// SIMATIC STEP 7 (V5.x) project Сварная машина 1
// CPU: CPU 316-2 DP
// station: Hardware
// station: SIMATIC 300(1)
// station: P_ADR_BUS
// station: P_ADR_BUS
// station: Configuration

SYMBOL_TABLE
"C1"	C 1	COUNTER	// Счетчик единиц
"C2"	C 2	COUNTER	// Счетчик тысяч
"C3"	C 3	COUNTER	// Счетчик миллионов
"FC1"	FC 1	FC 1	// Блокировки
"FC2"	FC 2	FC 2	// Управление транспортерами и вентиляторами
"FC3"	FC 3	FC 3	// Муфта
"FC4"	FC 4	FC 4	// Протяжка проволоки
"FC5"	FC 5	FC 5	// Регулировка скорости
"FC6"	FC 6	FC 6	// Привод сварной машины
"FC7"	FC 7	FC 7
"FC10"	FC 10	FC 10	// Сообщения
"FC11"	FC 11	FC 11	// Счетчик произведенной продукции.
"B8.3"	I 0.0	BOOL	// Заднее положение толкателей корпусов
"B8.4"	I 0.1	BOOL	// Магазин бланков пуст
"B8.5"	I 0.2	BOOL	// Обрыв проволоки с катушки
"B8.6"	I 0.3	BOOL	// ?
"LAK"	I 0.5	BOOL	// Контроль работы лакировки
"F1.1 - F1.2"	I 0.6	BOOL	// Тепловая защита привод.двигателя и вакуум.насоса
"K7.1"	I 0.7	BOOL	// Сушильная печь включена
"B12.1"	I 1.0	BOOL	// Профилирование минус
"B12.2"	I 1.1	BOOL	// Профилирование -15%
"B12.3"	I 1.2	BOOL	// Профилирование -5%
"B12.4"	I 1.3	BOOL	// Профилирование -синхронная скорость
"B12.5"	I 1.4	BOOL	// Профилирование +5%
"B12.6"	I 1.5	BOOL	// Профилирование +15%
"B12.7"	I 1.6	BOOL	// Профилирование плюс
"B8.1"	I 1.7	BOOL	// Счетчик готовой продукции
"B12.8"	I 2.0	BOOL	// Сечка плюс
"B12.9"	I 2.1	BOOL	// Сечка +15%
"B12.10"	I 2.2	BOOL	// Сечка +5%
"B12.11"	I 2.3	BOOL	// Сечка синхронно
"B12.12"	I 2.4	BOOL	// Сечка -5%
"B12.13"	I 2.5	BOOL	// Сечка -15%
"B12.14"	I 2.6	BOOL	// Сечка минус
"P2.3"	I 4.0	BOOL	// Темп. контура №1 больше нормы
"P2.4"	I 4.1	BOOL	// Темп. контура №2 больше нормы
"P2.5"	I 4.2	BOOL	// Темп. контура №3 больше нормы
"P2.6"	I 4.3	BOOL	// Темп. контура №4 больше нормы
"B1.1"	I 4.4	BOOL	// Давление контура №1 ниже нормы
"B1.2"	I 4.5	BOOL	// Давление контура №2 ниже нормы
"B1.3"	I 4.6	BOOL	// Давление контура №3 ниже нормы
"B1.4"	I 4.7	BOOL	// Давление контура №4 ниже нормы
"B1.5"	I 5.0	BOOL	// Давление воздуха
"S1.1, S1.2, S1.9"	I 5.1	BOOL	// Муфты, желоб.
"S1.3"	I 5.2	BOOL	// Магазин открыт
"S1.4"	I 5.3	BOOL	// Верхний электрод поднят
"S1.5"	I 5.4	BOOL	// Штурвал ручной прокрутки.
"S1.6"	I 5.5	BOOL	// Транспортный лоток
"S1.7"	I 5.6	BOOL	// Вальцы.
"S1.8"	I 5.7	BOOL	// Защитный экран.
"S3.1"	I 8.0	BOOL	// Приводной двигатель ВКЛ.
"S3.2"	I 8.1	BOOL	// Приводной двигатель ОТКЛ.
"S3.3"	I 8.2	BOOL	// Муфта(пульт) ВКЛ.
"S3.4"	I 8.3	BOOL	// Муфта(машина) ВКЛ.
"S3.5 - S3.6"	I 8.4	BOOL	// Муфта(пульт,машина) ОТКЛ.
"S3.7"	I 8.5	BOOL	// Подача бланков(пульт) ВКЛ. Вакуум.
"S3.8"	I 8.6	BOOL	// Подача бланков(машина) ВКЛ. Вакуум.
"S3.9 - S3.10"	I 8.7	BOOL	// Подача бланков(пульт,машина) ОТКЛ. Вакуум.
"S3.11"	I 9.0	BOOL	// Протяжка проволоки в ручном режиме ВКЛ.
"S3.12"	I 9.1	BOOL	// Протяжка проволоки в ручном режиме ОТКЛ.
"S3.13"	I 9.2	BOOL	// Электродвигатель профилирования ВКЛ.
"S3.14"	I 9.3	BOOL	// Электродвигатель сечки ВКЛ.
"S3.15"	I 9.4	BOOL	// Сброс
"S3.16"	I 9.5	BOOL	// КнопкаСТОП(пульт)
"S3.18"	I 9.6	BOOL	// Привод (Jog)
"S4.1"	I 9.7	BOOL	// Переключатель(замкнут-РУЧНОЕ, разомкнут-АВТОМАТ)
"M0.0"	M 0.0	BOOL	// Меркер СТОП
"M0.1"	M 0.1	BOOL	// Меркер температуры
"M0.2"	M 0.2	BOOL	// Меркер давления воды
"M0.3"	M 0.3	BOOL	// Меркер блокировок
"M0.4"	M 0.4	BOOL	// Меркер защиты
"M0.5"	M 0.5	BOOL	// Меркер АВАРИЯ
"M1.0"	M 1.0	BOOL	// Меркер протяжки проволоки.
"m10.0"	M 10.0	BOOL	// Тригер включения транспортеров
"m10.1"	M 10.1	BOOL	// Тригер включения вытяжного вентилятора
"m10.2"	M 10.2	BOOL	// Тригер включения лакировочных роликов
"m10.3"	M 10.3	BOOL	// Тригер включения муфты (Ручной режим)
"m10.4"	M 10.4	BOOL	// Тригер включения эл.муфты (Автом. режим)
"m11.0"	M 11.0	BOOL	// Тригер эл.двиг. профилирования (Jog)
"m11.1"	M 11.1	BOOL	// Тригер включения эл.двиг. сечки (Jog)
"m11.2"	M 11.2	BOOL	// Тригер включения привода (Jog)
"m11.3"	M 11.3	BOOL	// Тригер включения протяжки проволоки в ручном режиме
"M12.0"	M 12.0	BOOL	// Тригер включения основного привода
"M12.1"	M 12.1	BOOL	// Тригер включения эл.муфты (Автомат. режим)
"M14.0"	M 14.0	BOOL	// Тригер включения вакуума
"m15.0"	M 15.0	BOOL	// Меркер счета единиц
"m15.1"	M 15.1	BOOL	// Меркер счета тысяч
"М15.2"	M 15.2	BOOL	// Меркер счета миллионов
"M15.3"	M 15.3	BOOL	// Сброс счетчика готовой продукции
"M15.4"	M 15.4	BOOL	// Меркер сброса счетчика С1
"M15.5"	M 15.5	BOOL	// Меркер сброса счетчика С2
"M15.6"	M 15.6	BOOL	// Меркер сброса счетчика С3
"КН1"	M 200.0	BOOL	// Кнопка ПУСК транспортеров №1, №2
"КН2"	M 200.1	BOOL	// Кнопка СТОП транспортеров №1, №2
"КН3"	M 200.2	BOOL	// Кнопка ПУСК вытяжного вентилятора
"Кн4"	M 200.3	BOOL	// Кнопка СТОП вытяжного вентилятора
"Кн5"	M 200.4	BOOL	// Кнопка ПУСК лакировки
"Кн6"	M 200.5	BOOL	// Кнопка СТОП лакировки
"M2.1"	Q 12.0	BOOL	// Приводной двигатель.
"M2.1{Jog}"	Q 12.1	BOOL	// Привод (Jog)
"M3.2"	Q 12.3	BOOL	// Верхний электрод(привод) ВКЛ.
"M3.2 {MI1}"	Q 12.4	BOOL	// Электрод работа в ручном режиме
"M13.1"	Q 12.6	BOOL	// Транспорт. №1
"M13.2"	Q 12.7	BOOL	// Транспорт. №2
"M3.1"	Q 16.0	BOOL	// Электродвигатель профилирования.
"M3.1{Jog}"	Q 16.1	BOOL	// Профилирование{JOG}
"M3.1{-15}"	Q 16.2	BOOL	// Профилирование {-15}
"M3.1{-5}"	Q 16.3	BOOL	// Профилирование {-5}
"M3.1{0}"	Q 16.4	BOOL	// Профилирование {0}
"M3.1{+5}"	Q 16.5	BOOL	// Профилирование {+5}
"M3.1{+15}"	Q 16.6	BOOL	// Профилирование {+15}
"M3.3"	Q 20.0	BOOL	// Электродвигатель сечки.
"M3.3{MI1}"	Q 20.1	BOOL	// Сечка работа в ручном режиме
"M3.3{MI2}"	Q 20.2	BOOL	// Сечка{MI2}
"M3.3{MI3}"	Q 20.3	BOOL	// Сечка{MI3}
"M3.3{MI4}"	Q 20.4	BOOL	// Сечка{MI4}
"M3.3{JOG}"	Q 20.5	BOOL	// Сечка{JOG}
"M13.4"	Q 20.7	BOOL	// Наружный лак. ролик
"K9.4"	Q 24.0	BOOL	// Внутренний лак. ролик М13.3
"K9.2"	Q 24.1	BOOL	// Вытяжной вентилятор
"K9.3"	Q 24.4	BOOL	// Вакуум ВКЛ.
"K9.1"	Q 24.5	BOOL	// Эл.муфта
"T1"	T 1	TIMER	// Таймер задержки вкл. муфты
END_SYMBOL_TABLE

FUNCTION "FC1" : VOID	// FC 1
VERSION : 0.1
BEGIN
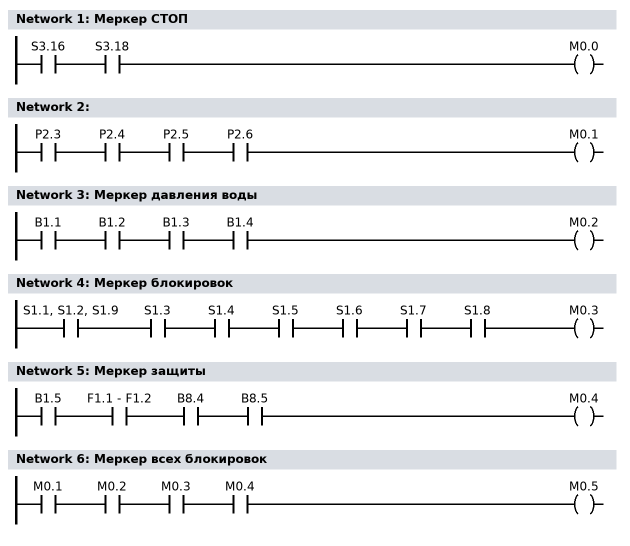
NETWORK
TITLE = Меркер СТОП
      A     "S3.16";
      A     "S3.18";
      =     "M0.0";
NETWORK
TITLE =
//Температура охлаждающей воды.
      A     "P2.3";
      A     "P2.4";
      A     "P2.5";
      A     "P2.6";
      =     "M0.1";
NETWORK
TITLE = Меркер давления воды
//Давление охлаждающей воды.
      A     "B1.1";
      A     "B1.2";
      A     "B1.3";
      A     "B1.4";
      =     "M0.2";
NETWORK
TITLE = Меркер блокировок
//Состояние блокировочных концевиков.
      A     "S1.1, S1.2, S1.9";
      A     "S1.3";
      A     "S1.4";
      A     "S1.5";
      A     "S1.6";
      A     "S1.7";
      A     "S1.8";
      =     "M0.3";
NETWORK
TITLE = Меркер защиты
//Контроль давления воздуха и тепловая защита.
      A     "B1.5";
      A     "F1.1 - F1.2";
      A     "B8.4";
      A     "B8.5";
      =     "M0.4";
NETWORK
TITLE = Меркер всех блокировок
      A     "M0.1";
      A     "M0.2";
      A     "M0.3";
      A     "M0.4";
      =     "M0.5";
END_FUNCTION

FUNCTION "FC2" : VOID	// FC 2
TITLE = Управление транспортерами и вентиляторами.
VERSION : 0.1
BEGIN
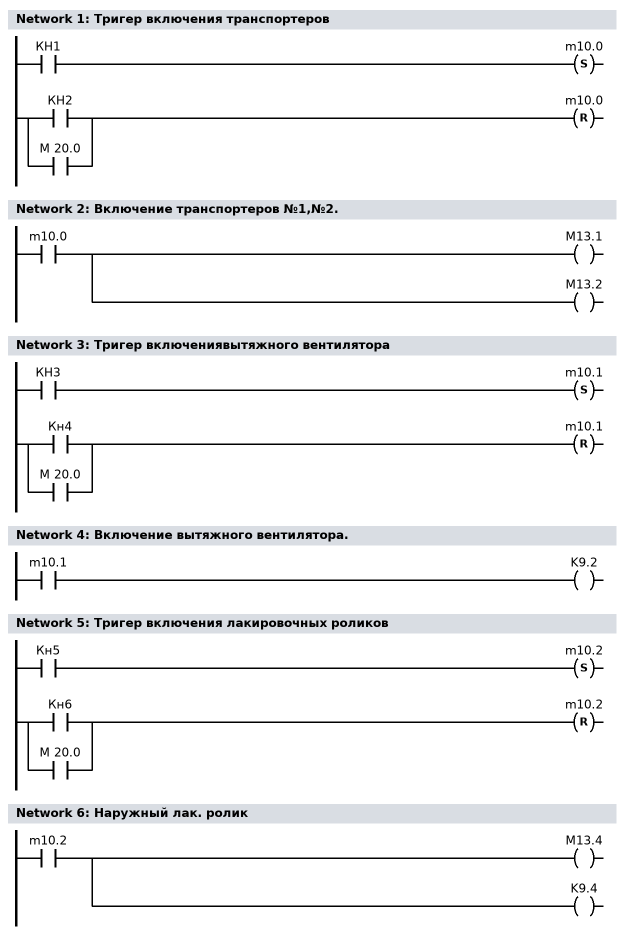
NETWORK
TITLE = Тригер включения транспортеров
      A     "КН1";
      S     "m10.0";
      A(;
      O     "КН2";
      O     M 20.0;
      );
      R     "m10.0";
      NOP   0;
NETWORK
TITLE = Включение транспортеров №1,№2.
      A     "m10.0";
      =     "M13.1";
      =     "M13.2";
NETWORK
TITLE = Тригер включениявытяжного вентилятора
      A     "КН3";
      S     "m10.1";
      A(;
      O     "Кн4";
      O     M 20.0;
      );
      R     "m10.1";
      NOP   0;
NETWORK
TITLE = Включение вытяжного вентилятора.
      A     "m10.1";
      =     "K9.2";
NETWORK
TITLE = Тригер включения лакировочных роликов
      A     "Кн5";
      S     "m10.2";
      A(;
      O     "Кн6";
      O     M 20.0;
      );
      R     "m10.2";
      NOP   0;
NETWORK
TITLE = Наружный лак. ролик
      A     "m10.2";
      =     "M13.4";
      =     "K9.4";
END_FUNCTION

FUNCTION "FC3" : VOID	// FC 3
TITLE = Муфта
//Включение муфты в ручном и автоматическом режимах.
VERSION : 0.1
BEGIN
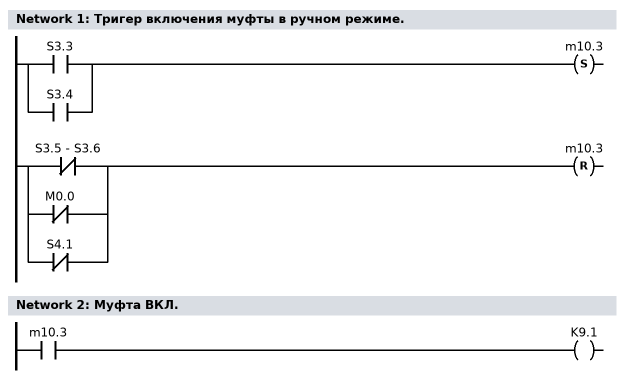
NETWORK
TITLE = Тригер включения муфты в ручном режиме.
      A(;
      O     "S3.3";
      O     "S3.4";
      );
      S     "m10.3";
      A(;
      ON    "S3.5 - S3.6";
      ON    "M0.0";
      ON    "S4.1";
      );
      R     "m10.3";
      NOP   0;
NETWORK
TITLE = Муфта ВКЛ.
//Включение муфты.
      A     "m10.3";
      =     "K9.1";
END_FUNCTION

FUNCTION "FC4" : VOID	// FC 4
TITLE = Протяжка проволоки.
VERSION : 0.1
BEGIN
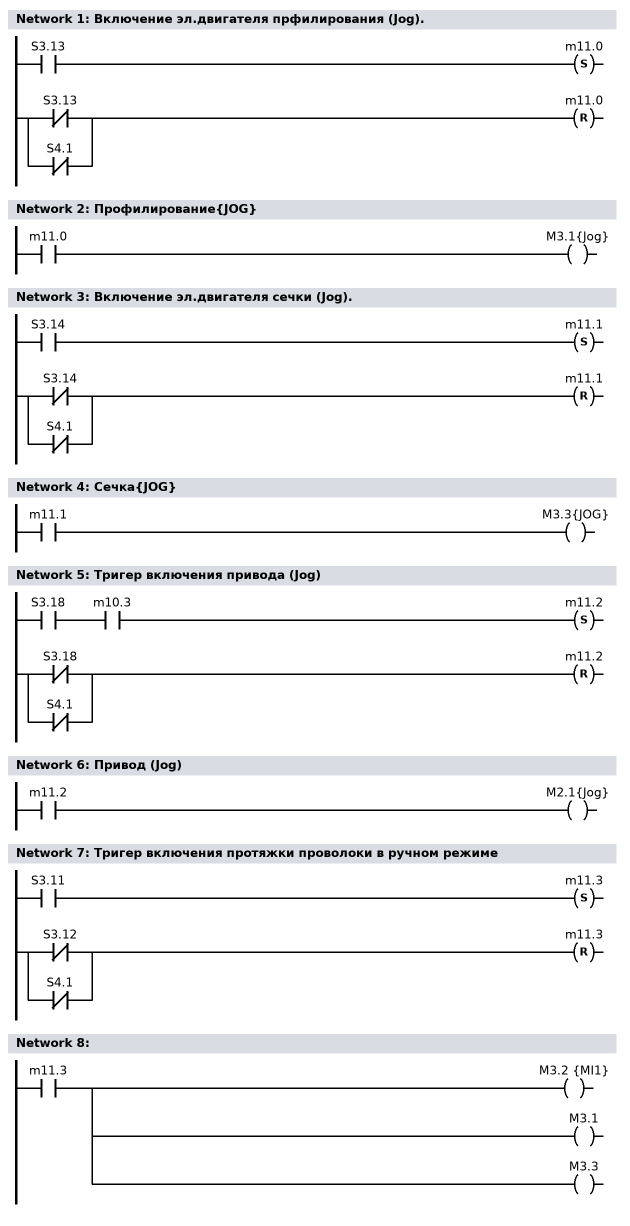
NETWORK
TITLE = Включение эл.двигателя прфилирования (Jog).
      A     "S3.13";
      S     "m11.0";
      A(;
      ON    "S3.13";
      ON    "S4.1";
      );
      R     "m11.0";
      NOP   0;
NETWORK
TITLE = Профилирование{JOG}
      A     "m11.0";
      =     "M3.1{Jog}";
NETWORK
TITLE = Включение эл.двигателя сечки (Jog).
      A     "S3.14";
      S     "m11.1";
      A(;
      ON    "S3.14";
      ON    "S4.1";
      );
      R     "m11.1";
      NOP   0;
NETWORK
TITLE = Сечка{JOG}
      A     "m11.1";
      =     "M3.3{JOG}";
NETWORK
TITLE = Тригер включения привода (Jog)
      A     "S3.18";
      A     "m10.3";
      S     "m11.2";
      A(;
      ON    "S3.18";
      ON    "S4.1";
      );
      R     "m11.2";
      NOP   0;
NETWORK
TITLE = Привод (Jog)
      A     "m11.2";
      =     "M2.1{Jog}";
NETWORK
TITLE = Тригер включения протяжки проволоки в ручном режиме
      A     "S3.11";
      S     "m11.3";
      A(;
      ON    "S3.12";
      ON    "S4.1";
      );
      R     "m11.3";
      NOP   0;
NETWORK
TITLE =
      A     "m11.3";
      =     "M3.2 {MI1}";
      =     "M3.1";
      =     "M3.3";
END_FUNCTION

FUNCTION "FC5" : VOID	// FC 5
TITLE = Регулирование скорости профилирования.
//Регулирование скорости эл.дв. профилирования при прямой подаче упр. сигнала с 
//аналогового выхода ЧП электрода на аналоговый вход ЧП профилирования.
VERSION : 0.1
BEGIN
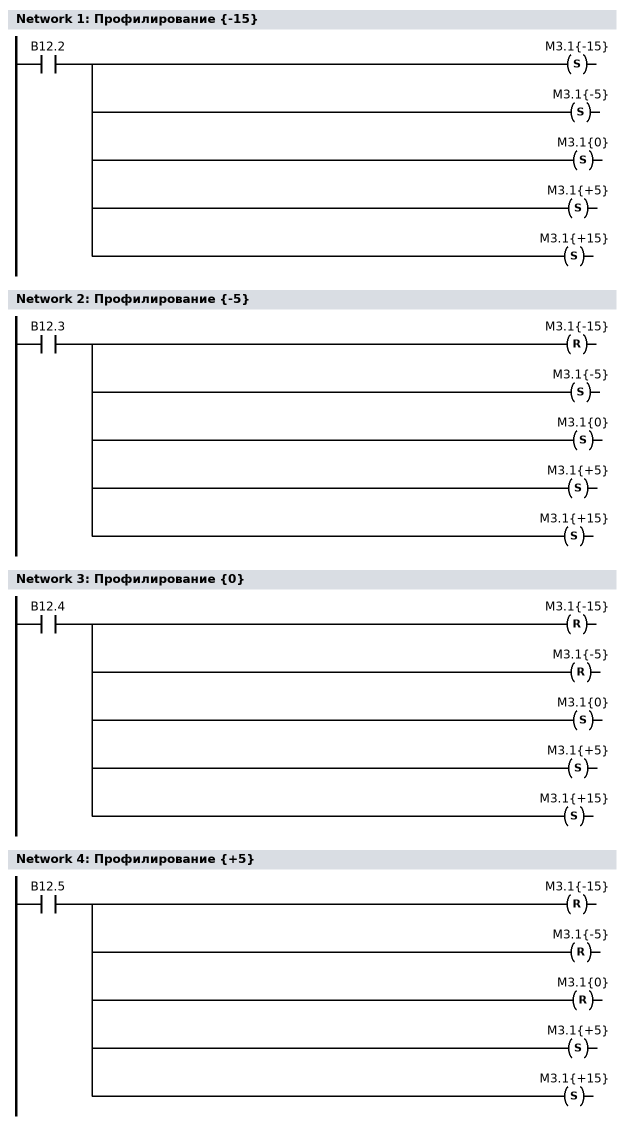
NETWORK
TITLE = Профилирование {-15}
      A     "B12.2";
      S     "M3.1{-15}";
      S     "M3.1{-5}";
      S     "M3.1{0}";
      S     "M3.1{+5}";
      S     "M3.1{+15}";
NETWORK
TITLE = Профилирование {-5}
      A     "B12.3";
      R     "M3.1{-15}";
      S     "M3.1{-5}";
      S     "M3.1{0}";
      S     "M3.1{+5}";
      S     "M3.1{+15}";
NETWORK
TITLE = Профилирование {0}
      A     "B12.4";
      R     "M3.1{-15}";
      R     "M3.1{-5}";
      S     "M3.1{0}";
      S     "M3.1{+5}";
      S     "M3.1{+15}";
NETWORK
TITLE = Профилирование {+5}
      A     "B12.5";
      R     "M3.1{-15}";
      R     "M3.1{-5}";
      R     "M3.1{0}";
      S     "M3.1{+5}";
      S     "M3.1{+15}";
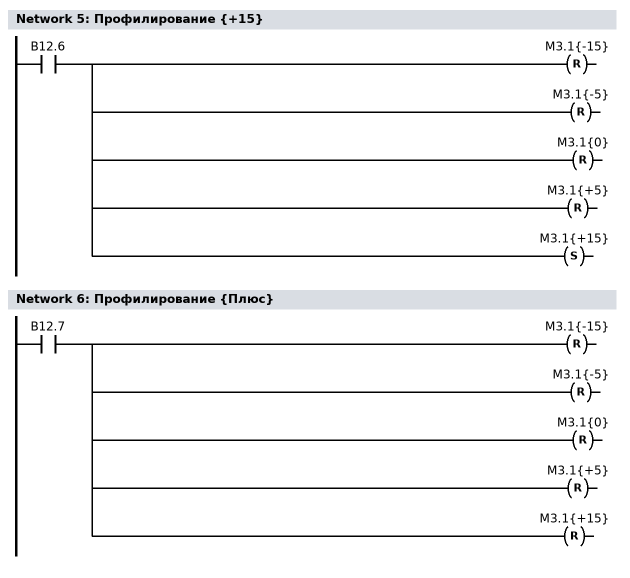
NETWORK
TITLE = Профилирование {+15}
      A     "B12.6";
      R     "M3.1{-15}";
      R     "M3.1{-5}";
      R     "M3.1{0}";
      R     "M3.1{+5}";
      S     "M3.1{+15}";
NETWORK
TITLE = Профилирование {Плюс}
      A     "B12.7";
      R     "M3.1{-15}";
      R     "M3.1{-5}";
      R     "M3.1{0}";
      R     "M3.1{+5}";
      R     "M3.1{+15}";
END_FUNCTION

FUNCTION "FC6" : VOID	// FC 6
TITLE = Привод сварной машины.
//Работа сварной машины в автоматическом режиме.
VERSION : 0.1
BEGIN
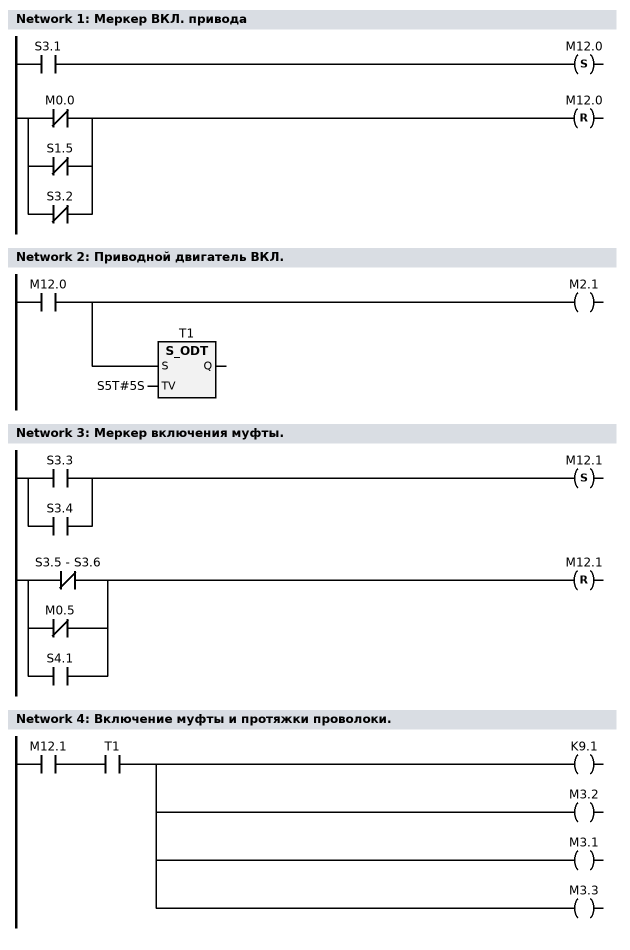
NETWORK
TITLE = Меркер ВКЛ. привода
      A     "S3.1";
      S     "M12.0";
      A(;
      ON    "M0.0";
      ON    "S1.5";
      ON    "S3.2";
      );
      R     "M12.0";
      NOP   0;
NETWORK
TITLE = Приводной двигатель ВКЛ.
      A     "M12.0";
      =     L 0.0;
      A     L 0.0;
      BLD   102;
      =     "M2.1";
      A     L 0.0;
      L     S5T#5S;
      SD    "T1";
      NOP   0;
      NOP   0;
      NOP   0;
      NOP   0;
NETWORK
TITLE = Меркер включения муфты.
      A(;
      O     "S3.3";
      O     "S3.4";
      );
      S     "M12.1";
      A(;
      ON    "S3.5 - S3.6";
      ON    "M0.5";
      O     "S4.1";
      );
      R     "M12.1";
      NOP   0;
NETWORK
TITLE = Включение муфты и протяжки проволоки.
      A     "M12.1";
      A     "T1";
      =     "K9.1";
      =     "M3.2";
      =     "M3.1";
      =     "M3.3";
END_FUNCTION

FUNCTION "FC7" : VOID	// FC 7
TITLE = Блок управления вакуумным насосом.
VERSION : 0.1
BEGIN
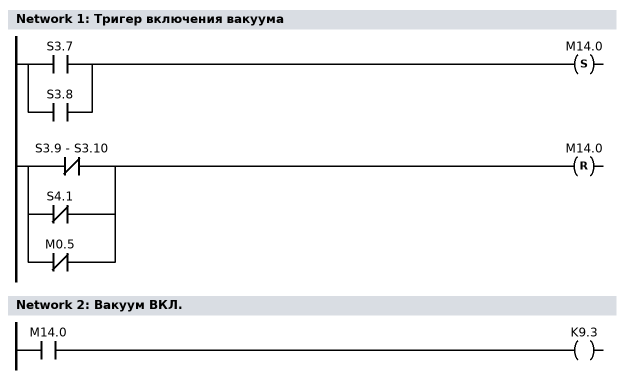
NETWORK
TITLE = Тригер включения вакуума
      A(;
      O     "S3.7";
      O     "S3.8";
      );
      S     "M14.0";
      A(;
      ON    "S3.9 - S3.10";
      ON    "S4.1";
      ON    "M0.5";
      );
      R     "M14.0";
      NOP   0;
NETWORK
TITLE = Вакуум ВКЛ.
      A     "M14.0";
      =     "K9.3";
END_FUNCTION

FUNCTION "FC10" : VOID	// FC 10
TITLE = Сообщения.
VERSION : 0.1
BEGIN
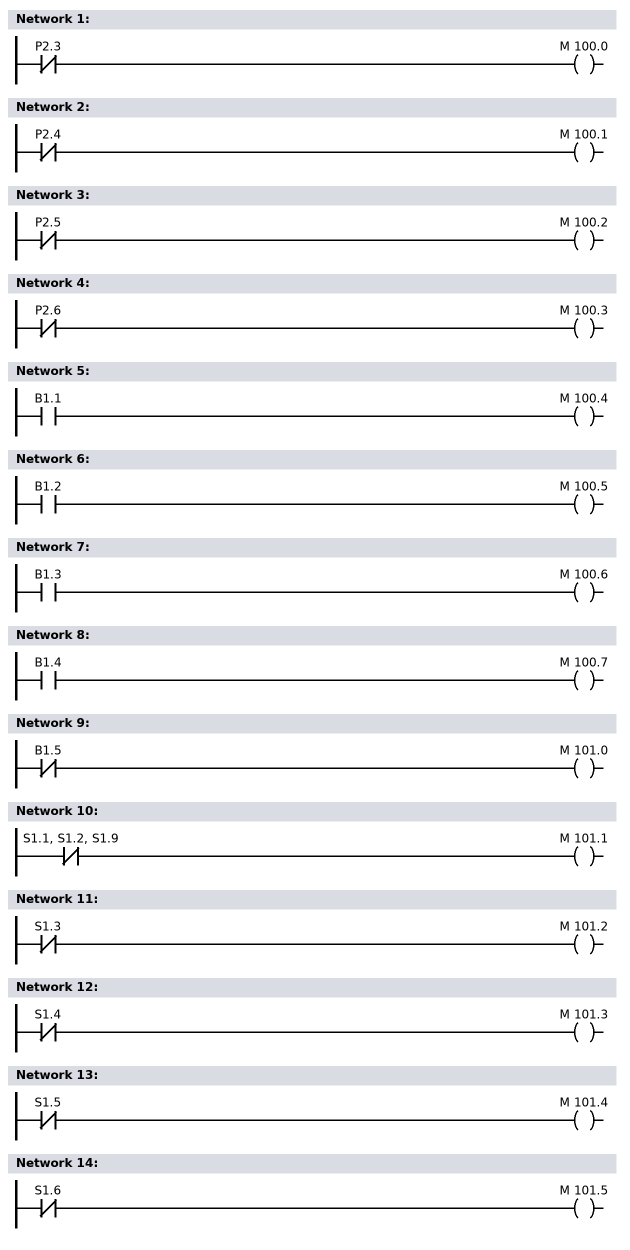
NETWORK
TITLE =
//Сообщение: Температура сварочного трансформатора выше нормы.
      AN    "P2.3";
      =     M 100.0;
NETWORK
TITLE =
//Сообщение: Температура нижнего электрода выше нормы.
      AN    "P2.4";
      =     M 100.1;
NETWORK
TITLE =
//Сообщение: Температура верхнего электрода выше нормы.
      AN    "P2.5";
      =     M 100.2;
NETWORK
TITLE =
//ообщение: Температура шибера выше нормы.
      AN    "P2.6";
      =     M 100.3;
NETWORK
TITLE =
//Сообщение: Проток охлаждающей воды в трансформаторе ниже нормы.
      A     "B1.1";
      =     M 100.4;
NETWORK
TITLE =
//Сообщение: Проток охлаждающей воды нижнего электрода ниже нормы.
      A     "B1.2";
      =     M 100.5;
NETWORK
TITLE =
//Сообщение: Проток охлаждающей воды верхнего электрода ниже нормы.
      A     "B1.3";
      =     M 100.6;
NETWORK
TITLE =
//Сообщение: Проток охлаждающей воды шибера ниже нормы.
      A     "B1.4";
      =     M 100.7;
NETWORK
TITLE =
//Сообщение: Нет воздуха.
      AN    "B1.5";
      =     M 101.0;
NETWORK
TITLE =
//Сообщение: Муфта и .......
      AN    "S1.1, S1.2, S1.9";
      =     M 101.1;
NETWORK
TITLE =
//Сообщение: Магазин бланков открыт.
      AN    "S1.3";
      =     M 101.2;
NETWORK
TITLE =
//Сообщение: Верхний электрод поднят.
      AN    "S1.4";
      =     M 101.3;
NETWORK
TITLE =
//Сообщение: Штурвал в режиме прокрутки.
      AN    "S1.5";
      =     M 101.4;
NETWORK
TITLE =
      AN    "S1.6";
      =     M 101.5;
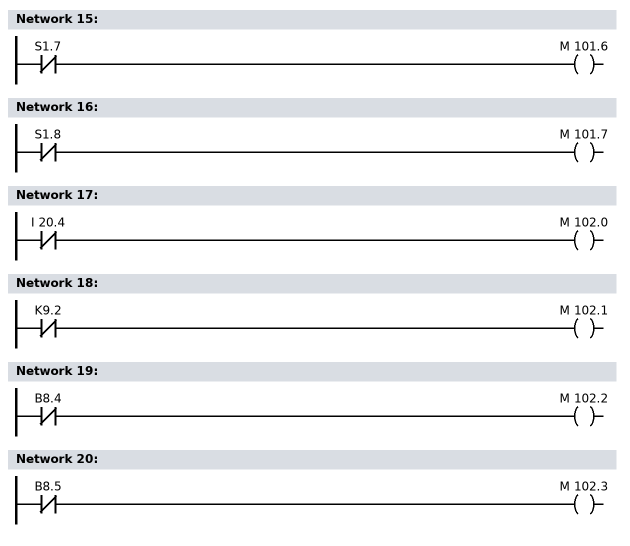
NETWORK
TITLE =
      AN    "S1.7";
      =     M 101.6;
NETWORK
TITLE =
      AN    "S1.8";
      =     M 101.7;
NETWORK
TITLE =
      AN    I 20.4;
      =     M 102.0;
NETWORK
TITLE =
      AN    "K9.2";
      =     M 102.1;
NETWORK
TITLE =
      AN    "B8.4";
      =     M 102.2;
NETWORK
TITLE =
      AN    "B8.5";
      =     M 102.3;
END_FUNCTION

FUNCTION "FC11" : VOID	// FC 11
TITLE = Счетчик произведенной продукции.
VERSION : 0.1
BEGIN
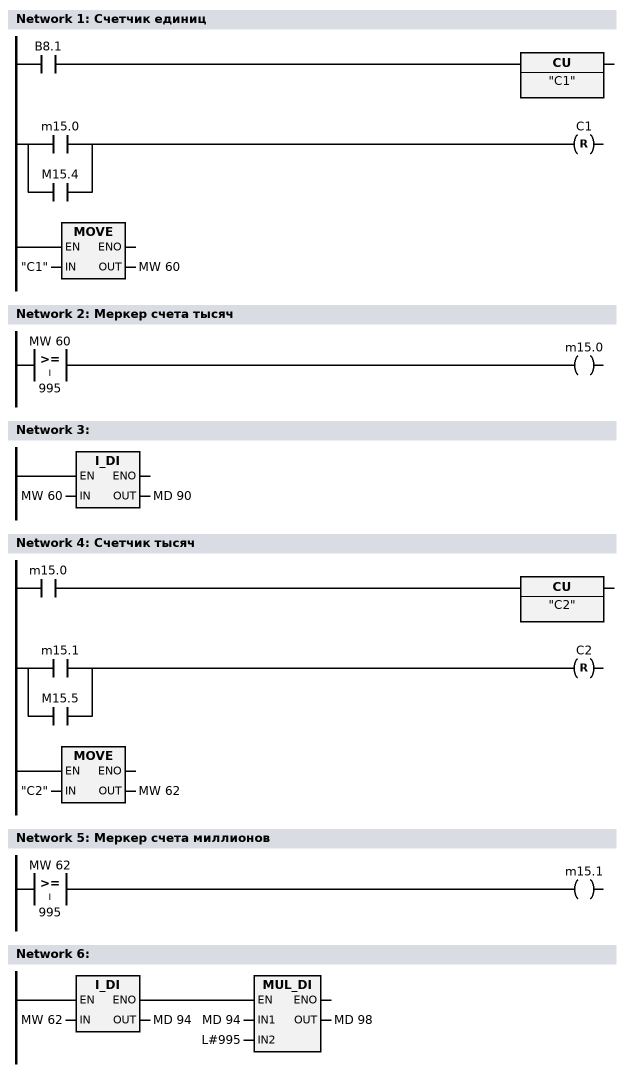
NETWORK
TITLE = Счетчик единиц
      A     "B8.1";
      CU    "C1";
      BLD   101;
      NOP   0;
      NOP   0;
      A(;
      O     "m15.0";
      O     "M15.4";
      );
      R     "C1";
      L     "C1";
      T     MW 60;
      NOP   0;
      NOP   0;
NETWORK
TITLE = Меркер счета тысяч
      L     MW 60;
      L     995;
      >=I;
      =     "m15.0";
NETWORK
TITLE =
      L     MW 60;
      ITD;
      T     MD 90;
      NOP   0;
NETWORK
TITLE = Счетчик тысяч
      A     "m15.0";
      CU    "C2";
      BLD   101;
      NOP   0;
      NOP   0;
      A(;
      O     "m15.1";
      O     "M15.5";
      );
      R     "C2";
      L     "C2";
      T     MW 62;
      NOP   0;
      NOP   0;
NETWORK
TITLE = Меркер счета миллионов
      L     MW 62;
      L     995;
      >=I;
      =     "m15.1";
NETWORK
TITLE =
      A(;
      L     MW 62;
      ITD;
      T     MD 94;
      SET;
      SAVE;
      CLR;
      A     BR;
      );
      JNB   _001;
      L     MD 94;
      L     L#995;
      *D;
      T     MD 98;
_001: NOP   0;
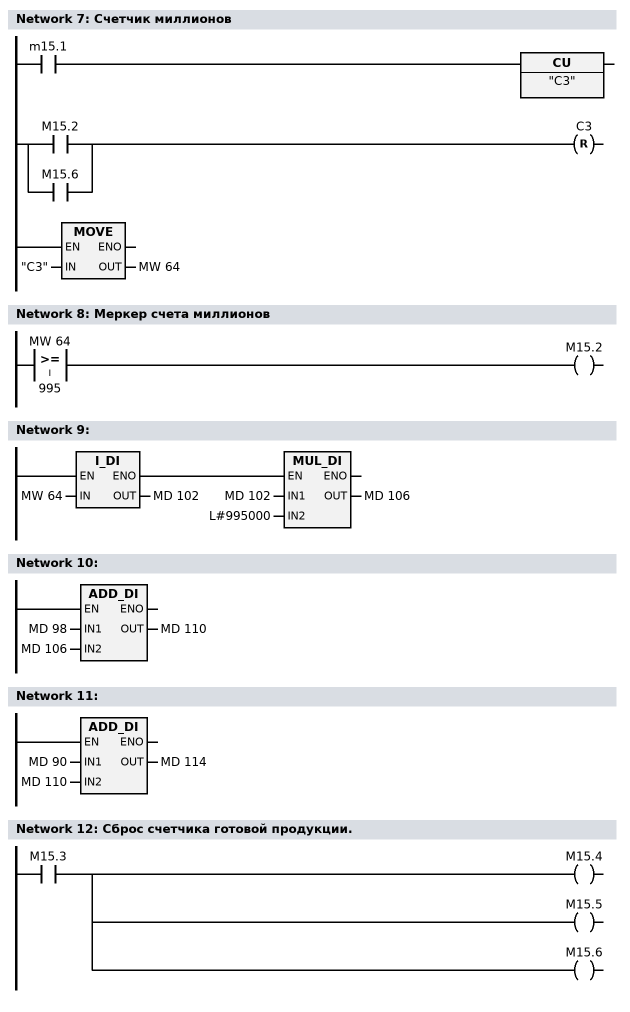
NETWORK
TITLE = Счетчик миллионов
      A     "m15.1";
      CU    "C3";
      BLD   101;
      NOP   0;
      NOP   0;
      A(;
      O     "М15.2";
      O     "M15.6";
      );
      R     "C3";
      L     "C3";
      T     MW 64;
      NOP   0;
      NOP   0;
NETWORK
TITLE = Меркер счета миллионов
      L     MW 64;
      L     995;
      >=I;
      =     "М15.2";
NETWORK
TITLE =
      A(;
      L     MW 64;
      ITD;
      T     MD 102;
      SET;
      SAVE;
      CLR;
      A     BR;
      );
      JNB   _002;
      L     MD 102;
      L     L#995000;
      *D;
      T     MD 106;
_002: NOP   0;
NETWORK
TITLE =
      L     MD 98;
      L     MD 106;
      +D;
      T     MD 110;
      NOP   0;
NETWORK
TITLE =
      L     MD 90;
      L     MD 110;
      +D;
      T     MD 114;
      NOP   0;
NETWORK
TITLE = Сброс счетчика готовой продукции.
      A     "M15.3";
      =     "M15.4";
      =     "M15.5";
      =     "M15.6";
END_FUNCTION

ORGANIZATION_BLOCK OB 1
TITLE = "Main Program Sweep (Cycle)"
VERSION : 0.1
VAR_TEMP
  OB1_EV_CLASS : BYTE ;	//Bits 0-3 = 1 (Coming event), Bits 4-7 = 1 (Event class 1)
  OB1_SCAN_1 : BYTE ;	//1 (Cold restart scan 1 of OB 1), 3 (Scan 2-n of OB 1)
  OB1_PRIORITY : BYTE ;	//Priority of OB Execution
  OB1_OB_NUMBR : BYTE ;	//1 (Organization block 1, OB1)
  OB1_RESERVED_1 : BYTE ;	//Reserved for system
  OB1_RESERVED_2 : BYTE ;	//Reserved for system
  OB1_PREV_CYCLE : INT ;	//Cycle time of previous OB1 scan (milliseconds)
  OB1_MIN_CYCLE : INT ;	//Minimum cycle time of OB1 (milliseconds)
  OB1_MAX_CYCLE : INT ;	//Maximum cycle time of OB1 (milliseconds)
  OB1_DATE_TIME : DATE_AND_TIME ;	//Date and time OB1 started
END_VAR
BEGIN
NETWORK
TITLE =
      UC    "FC1";
NETWORK
TITLE =
      UC    "FC2";
NETWORK
TITLE =
      UC    "FC3";
NETWORK
TITLE =
      UC    "FC4";
NETWORK
TITLE =
      UC    "FC5";
NETWORK
TITLE =
      UC    "FC6";
NETWORK
TITLE =
      UC    "FC10";
NETWORK
TITLE =
      UC    "FC11";
END_ORGANIZATION_BLOCK
